(* IEC 61131-3 sources: volt/packages/volt-lsp-iec/test-corpus/pro2193/Device/Plc Logic/Application/99 Library/Functions/CONCAT, 14 files *)

(* ---- CONCAT3.pou ---- *)
// Concatenates 3 strings
FUNCTION CONCAT3 : STRING(255)
VAR_INPUT
	s1	: STRING(255);
	s2	: STRING(255);
	s3	: STRING(255);
END_VAR

%LANGUAGE ST
Stu.StrCpyA(
	pBuffer		:= ADR(CONCAT3),
	iBufferSize	:= 255,
	pStr		:= ADR(s1));

IF	Stu.StrConcatA(pstFrom := ADR(s2), pstTo := ADR(CONCAT3), iBufferSize := 255) THEN
	Stu.StrConcatA(pstFrom := ADR(s3), pstTo := ADR(CONCAT3), iBufferSize := 255);
END_IF

END_FUNCTION

(* ---- CONCAT4.pou ---- *)
// Concatenates 4 strings
FUNCTION CONCAT4 : STRING(255)
VAR_INPUT
	s1	: STRING(255);
	s2	: STRING(255);
	s3	: STRING(255);
	s4	: STRING(255);
END_VAR

%LANGUAGE ST
Stu.StrCpyA(
	pBuffer		:= ADR(CONCAT4),
	iBufferSize	:= 255,
	pStr		:= ADR(s1));

IF		Stu.StrConcatA(pstFrom := ADR(s2), pstTo := ADR(CONCAT4), iBufferSize := 255) THEN
	IF	Stu.StrConcatA(pstFrom := ADR(s3), pstTo := ADR(CONCAT4), iBufferSize := 255) THEN
		Stu.StrConcatA(pstFrom := ADR(s4), pstTo := ADR(CONCAT4), iBufferSize := 255);
	END_IF
END_IF

END_FUNCTION

(* ---- CONCAT5.pou ---- *)
// Concatenates 5 strings
FUNCTION CONCAT5 : STRING(255)
VAR_INPUT
	s1	: STRING(255);
	s2	: STRING(255);
	s3	: STRING(255);
	s4	: STRING(255);
	s5	: STRING(255);
END_VAR

%LANGUAGE ST
Stu.StrCpyA(
	pBuffer		:= ADR(CONCAT5),
	iBufferSize	:= 255,
	pStr		:= ADR(s1));

IF			Stu.StrConcatA(pstFrom := ADR(s2), pstTo := ADR(CONCAT5), iBufferSize := 255) THEN
	IF		Stu.StrConcatA(pstFrom := ADR(s3), pstTo := ADR(CONCAT5), iBufferSize := 255) THEN
		IF	Stu.StrConcatA(pstFrom := ADR(s4), pstTo := ADR(CONCAT5), iBufferSize := 255) THEN
			Stu.StrConcatA(pstFrom := ADR(s5), pstTo := ADR(CONCAT5), iBufferSize := 255);
		END_IF
	END_IF
END_IF

END_FUNCTION

(* ---- CONCAT6.pou ---- *)
// Concatenates 6 strings
FUNCTION CONCAT6 : STRING(255)
VAR_INPUT
	s1	: STRING(255);
	s2	: STRING(255);
	s3	: STRING(255);
	s4	: STRING(255);
	s5	: STRING(255);
	s6	: STRING(255);
END_VAR

%LANGUAGE ST
Stu.StrCpyA(
	pBuffer		:= ADR(CONCAT6),
	iBufferSize	:= 255,
	pStr		:= ADR(s1));

IF				Stu.StrConcatA(pstFrom := ADR(s2), pstTo := ADR(CONCAT6), iBufferSize := 255) THEN
	IF			Stu.StrConcatA(pstFrom := ADR(s3), pstTo := ADR(CONCAT6), iBufferSize := 255) THEN
		IF		Stu.StrConcatA(pstFrom := ADR(s4), pstTo := ADR(CONCAT6), iBufferSize := 255) THEN
			IF	Stu.StrConcatA(pstFrom := ADR(s5), pstTo := ADR(CONCAT6), iBufferSize := 255) THEN
				Stu.StrConcatA(pstFrom := ADR(s6), pstTo := ADR(CONCAT6), iBufferSize := 255);
			END_IF
		END_IF
	END_IF
END_IF

END_FUNCTION

(* ---- CONCAT7.pou ---- *)
// Concatenates 7 strings
FUNCTION CONCAT7 : STRING(255)
VAR_INPUT
	s1	: STRING(255);
	s2	: STRING(255);
	s3	: STRING(255);
	s4	: STRING(255);
	s5	: STRING(255);
	s6	: STRING(255);
	s7	: STRING(255);
END_VAR

%LANGUAGE ST
Stu.StrCpyA(
	pBuffer		:= ADR(CONCAT7),
	iBufferSize	:= 255,
	pStr		:= ADR(s1));

IF					Stu.StrConcatA(pstFrom := ADR(s2), pstTo := ADR(CONCAT7), iBufferSize := 255) THEN
	IF				Stu.StrConcatA(pstFrom := ADR(s3), pstTo := ADR(CONCAT7), iBufferSize := 255) THEN
		IF			Stu.StrConcatA(pstFrom := ADR(s4), pstTo := ADR(CONCAT7), iBufferSize := 255) THEN
			IF		Stu.StrConcatA(pstFrom := ADR(s5), pstTo := ADR(CONCAT7), iBufferSize := 255) THEN
				IF	Stu.StrConcatA(pstFrom := ADR(s6), pstTo := ADR(CONCAT7), iBufferSize := 255) THEN
					Stu.StrConcatA(pstFrom := ADR(s7), pstTo := ADR(CONCAT7), iBufferSize := 255);
				END_IF
			END_IF
		END_IF
	END_IF
END_IF

END_FUNCTION

(* ---- CONCAT8.pou ---- *)
// Concatenates 8 strings
FUNCTION CONCAT8 : STRING(255)
VAR_INPUT
	s1	: STRING(255);
	s2	: STRING(255);
	s3	: STRING(255);
	s4	: STRING(255);
	s5	: STRING(255);
	s6	: STRING(255);
	s7	: STRING(255);
	s8	: STRING(255);
END_VAR

%LANGUAGE ST
Stu.StrCpyA(
	pBuffer		:= ADR(CONCAT8),
	iBufferSize	:= 255,
	pStr		:= ADR(s1));

IF						Stu.StrConcatA(pstFrom := ADR(s2), pstTo := ADR(CONCAT8), iBufferSize := 255) THEN
	IF					Stu.StrConcatA(pstFrom := ADR(s3), pstTo := ADR(CONCAT8), iBufferSize := 255) THEN
		IF				Stu.StrConcatA(pstFrom := ADR(s4), pstTo := ADR(CONCAT8), iBufferSize := 255) THEN
			IF			Stu.StrConcatA(pstFrom := ADR(s5), pstTo := ADR(CONCAT8), iBufferSize := 255) THEN
				IF		Stu.StrConcatA(pstFrom := ADR(s6), pstTo := ADR(CONCAT8), iBufferSize := 255) THEN
					IF	Stu.StrConcatA(pstFrom := ADR(s7), pstTo := ADR(CONCAT8), iBufferSize := 255) THEN
						Stu.StrConcatA(pstFrom := ADR(s8), pstTo := ADR(CONCAT8), iBufferSize := 255);
					END_IF
				END_IF
			END_IF
		END_IF
	END_IF
END_IF

END_FUNCTION

(* ---- CONCAT9.pou ---- *)
// Concatenates 9 strings
FUNCTION CONCAT9 : STRING(255)
VAR_INPUT
	s1	: STRING(255);
	s2	: STRING(255);
	s3	: STRING(255);
	s4	: STRING(255);
	s5	: STRING(255);
	s6	: STRING(255);
	s7	: STRING(255);
	s8	: STRING(255);
	s9	: STRING(255);
END_VAR

%LANGUAGE ST
Stu.StrCpyA(
	pBuffer		:= ADR(CONCAT9),
	iBufferSize	:= 255,
	pStr		:= ADR(s1));

IF							Stu.StrConcatA(pstFrom := ADR(s2), pstTo := ADR(CONCAT9), iBufferSize := 255) THEN
	IF						Stu.StrConcatA(pstFrom := ADR(s3), pstTo := ADR(CONCAT9), iBufferSize := 255) THEN
		IF					Stu.StrConcatA(pstFrom := ADR(s4), pstTo := ADR(CONCAT9), iBufferSize := 255) THEN
			IF				Stu.StrConcatA(pstFrom := ADR(s5), pstTo := ADR(CONCAT9), iBufferSize := 255) THEN
				IF			Stu.StrConcatA(pstFrom := ADR(s6), pstTo := ADR(CONCAT9), iBufferSize := 255) THEN
					IF		Stu.StrConcatA(pstFrom := ADR(s7), pstTo := ADR(CONCAT9), iBufferSize := 255) THEN
						IF	Stu.StrConcatA(pstFrom := ADR(s8), pstTo := ADR(CONCAT9), iBufferSize := 255) THEN
							Stu.StrConcatA(pstFrom := ADR(s9), pstTo := ADR(CONCAT9), iBufferSize := 255);
						END_IF
					END_IF
				END_IF
			END_IF
		END_IF
	END_IF
END_IF

END_FUNCTION

(* ---- CONCATARRAY.pou ---- *)
// Concatenates any array of strings with optional separator between the strings
FUNCTION CONCATARRAY : STRING(255)
VAR_IN_OUT
	str					: ARRAY[*] OF STRING(255);
END_VAR
VAR_INPUT
	separator			: STRING(10)	:= '';	// Optional separator character between the string parts
END_VAR
VAR
	upper, lower, di	: DINT;
END_VAR

%LANGUAGE ST
lower		:= LOWER_BOUND(str, 1);
upper		:= UPPER_BOUND(str, 1);

CONCATARRAY	:= str[lower];

IF upper = lower THEN
	RETURN;
END_IF

FOR di := lower + 1 TO upper DO
	IF NOT Stu.StrConcatA(				// Add separator char
				pstFrom		:= ADR(separator),
				pstTo		:= ADR(CONCATARRAY),
				iBufferSize	:= 255)
	THEN
		RETURN;		// Stop concatenating the string when StrConcatA fails
	END_IF

	IF NOT Stu.StrConcatA(
				pstFrom		:= ADR(str[di]),
				pstTo		:= ADR(CONCATARRAY),
				iBufferSize	:= 255)
	THEN
		RETURN;		// Stop concatenating the string when StrConcatA fails
	END_IF
END_FOR

END_FUNCTION

(* ---- SAFECONCAT10.pou ---- *)
// Safely concatenates 10 strings
FUNCTION SAFECONCAT10 : BOOL
VAR_INPUT
	s1			: Stu.CharBufferPtr;	// Result string goes here
	s2			: STRING(80);			// First string to add
	s3			: STRING(80);			// Second string to add
	s4			: STRING(80);			// Third string to add
	s5			: STRING(80);			// Fourth string to add
	s6			: STRING(80);			// Fifth string to add
	s7			: STRING(80);			// xth string to add
	s8			: STRING(80);			// xth string to add
	s9			: STRING(80);			// xth string to add
	s10			: STRING(80);			// xth string to add
	bufferSize	: INT;					// bufferSize of s1
END_VAR

%LANGUAGE ST
IF												StrConcatA(pstFrom := ADR(s2), pstTo := s1, iBufferSize := bufferSize) THEN
	IF											StrConcatA(pstFrom := ADR(s3), pstTo := s1, iBufferSize := bufferSize) THEN
		IF										StrConcatA(pstFrom := ADR(s4), pstTo := s1, iBufferSize := bufferSize) THEN
			IF									StrConcatA(pstFrom := ADR(s5), pstTo := s1, iBufferSize := bufferSize) THEN
				IF								StrConcatA(pstFrom := ADR(s6), pstTo := s1, iBufferSize := bufferSize) THEN
					IF							StrConcatA(pstFrom := ADR(s7), pstTo := s1, iBufferSize := bufferSize) THEN
						IF						StrConcatA(pstFrom := ADR(s8), pstTo := s1, iBufferSize := bufferSize) THEN
							IF					StrConcatA(pstFrom := ADR(s9), pstTo := s1, iBufferSize := bufferSize) THEN
								SAFECONCAT10 :=	StrConcatA(pstFrom := ADR(s10), pstTo := s1, iBufferSize := bufferSize);
							END_IF
						END_IF
					END_IF
				END_IF
			END_IF
		END_IF
	END_IF
END_IF

END_FUNCTION

(* ---- SAFECONCAT2.pou ---- *)
// Safely concatenates 2 strings
FUNCTION SAFECONCAT2 : BOOL
VAR_INPUT
	s1			: Stu.CharBufferPtr;	// Result string goes here
	s2			: STRING(80);			// String to add
	bufferSize	: INT;					// bufferSize of s1
END_VAR

%LANGUAGE ST
SAFECONCAT2 := StrConcatA(pstFrom := ADR(s2), pstTo := s1, iBufferSize := bufferSize);

END_FUNCTION

(* ---- SAFECONCAT3.pou ---- *)
// Safely concatenates 3 strings
FUNCTION SAFECONCAT3 : BOOL
VAR_INPUT
	s1			: Stu.CharBufferPtr;	// Result string goes here
	s2			: STRING(80);			// First string to add
	s3			: STRING(80);			// Second string to add
	bufferSize	: INT;					// bufferSize of s1
END_VAR

%LANGUAGE ST
IF					StrConcatA(pstFrom := ADR(s2), pstTo := s1, iBufferSize := bufferSize) THEN
	SAFECONCAT3 :=	StrConcatA(pstFrom := ADR(s3), pstTo := s1, iBufferSize := bufferSize);
END_IF

END_FUNCTION

(* ---- SAFECONCAT4.pou ---- *)
// Safely concatenates 4 strings
FUNCTION SAFECONCAT4 : BOOL
VAR_INPUT
	s1			: Stu.CharBufferPtr;	// Result string goes here
	s2			: STRING(80);			// First string to add
	s3			: STRING(80);			// Second string to add
	s4			: STRING(80);			// Third string to add
	bufferSize	: INT;					// bufferSize of s1
END_VAR

%LANGUAGE ST
IF						StrConcatA(pstFrom := ADR(s2), pstTo := s1, iBufferSize := bufferSize) THEN
	IF					StrConcatA(pstFrom := ADR(s3), pstTo := s1, iBufferSize := bufferSize) THEN
		SAFECONCAT4 :=	StrConcatA(pstFrom := ADR(s4), pstTo := s1, iBufferSize := bufferSize);
	END_IF
END_IF

END_FUNCTION

(* ---- SAFECONCAT5.pou ---- *)
// Safely concatenates 5 strings
FUNCTION SAFECONCAT5 : BOOL
VAR_INPUT
	s1			: Stu.CharBufferPtr;	// Result string goes here
	s2			: STRING(80);			// First string to add
	s3			: STRING(80);			// Second string to add
	s4			: STRING(80);			// Third string to add
	s5			: STRING(80);			// Fourth string to add
	bufferSize	: INT;					// bufferSize of s1
END_VAR

%LANGUAGE ST
IF							StrConcatA(pstFrom := ADR(s2), pstTo := s1, iBufferSize := bufferSize) THEN
	IF						StrConcatA(pstFrom := ADR(s3), pstTo := s1, iBufferSize := bufferSize) THEN
		IF					StrConcatA(pstFrom := ADR(s4), pstTo := s1, iBufferSize := bufferSize) THEN
			SAFECONCAT5 :=	StrConcatA(pstFrom := ADR(s5), pstTo := s1, iBufferSize := bufferSize);
		END_IF
	END_IF
END_IF

END_FUNCTION

(* ---- SAFECONCAT6.pou ---- *)
// Safely concatenates 6 strings
FUNCTION SAFECONCAT6 : BOOL
VAR_INPUT
	s1			: Stu.CharBufferPtr;	// Result string goes here
	s2			: STRING(80);			// First string to add
	s3			: STRING(80);			// Second string to add
	s4			: STRING(80);			// Third string to add
	s5			: STRING(80);			// Fourth string to add
	s6			: STRING(80);			// Fifth string to add
	bufferSize	: INT;					// bufferSize of s1
END_VAR

%LANGUAGE ST
IF								StrConcatA(pstFrom := ADR(s2), pstTo := s1, iBufferSize := bufferSize) THEN
	IF							StrConcatA(pstFrom := ADR(s3), pstTo := s1, iBufferSize := bufferSize) THEN
		IF						StrConcatA(pstFrom := ADR(s4), pstTo := s1, iBufferSize := bufferSize) THEN
			IF					StrConcatA(pstFrom := ADR(s5), pstTo := s1, iBufferSize := bufferSize) THEN
				SAFECONCAT6 :=	StrConcatA(pstFrom := ADR(s6), pstTo := s1, iBufferSize := bufferSize);
			END_IF
		END_IF
	END_IF
END_IF

END_FUNCTION
